// TIA Portal V16 export
// export: Created 2022-08-03T14:37:58.543671Z, ExportSetting WithDefaults, DisplayName Totally Integrated Automation Portal, DisplayVersion V16, DisplayName TIA Portal Version Control Interface, DisplayVersion V16, DisplayName TIA Portal Openness, DisplayVersion V16, DisplayName SINAMICS Startdrive Advanced, DisplayVersion V16, DisplayName SINAMICS Startdrive G130, G150, S120, S150, SINAMICS MV, S210, DisplayVersion V16, DisplayName SINAMICS Startdrive G110M, G120, G120C, G120D, G120P, DisplayVersion V16, DisplayName STEP 7 Professional, DisplayVersion V16, DisplayName STEP 7 Safety, DisplayVersion V16, DisplayName WinCC Professional, DisplayVersion V16
ORGANIZATION_BLOCK "Electrical_interlock"   // OB1, LAD, ProgramCycle
TITLE = "Main Program Sweep (Cycle)"
{ S7_Optimized_Access := 'TRUE' }
VERSION : 0.1
// stored: AutoNumber true, IsIECCheckEnabled false, SetENOAutomatically false
   VAR_INPUT
      Initial_Call : Bool;   // Initial call of this OB
      Remanence : Bool;   // =True, if remanent data are available
   END_VAR
BEGIN

REGION Network 1
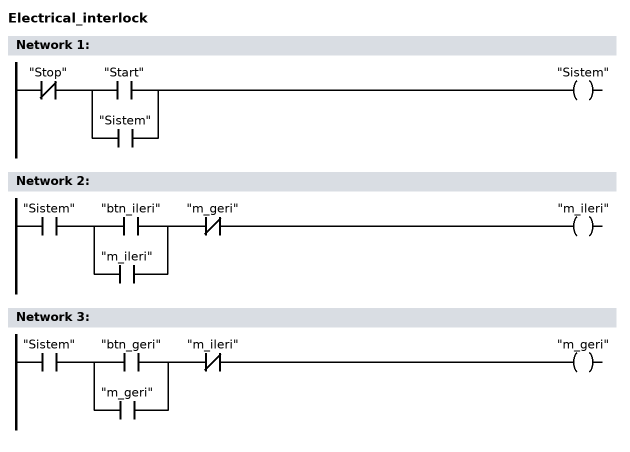
   RUNG wire#powerrail
      I_Contact( "Stop" )
      wire#w1
      Contact( "Start" )
      wire#w2
      Coil( "Sistem" )
   END_RUNG
   RUNG wire#w1
      Contact( "Sistem" )
   END_RUNG wire#w2
   // the same network as SCL:
   "Sistem" := NOT "Stop" AND ("Start" OR "Sistem");
END_REGION

REGION Network 2
   RUNG wire#powerrail
      Contact( "Sistem" )
      wire#w1
      Contact( "btn_ileri" )
      wire#w2
      I_Contact( "m_geri" )
      Coil( "m_ileri" )
   END_RUNG
   RUNG wire#w1
      Contact( "m_ileri" )
   END_RUNG wire#w2
   // the same network as SCL:
   "m_ileri" := "Sistem" AND ("btn_ileri" OR "m_ileri") AND NOT "m_geri";
END_REGION

REGION Network 3
   RUNG wire#powerrail
      Contact( "Sistem" )
      wire#w1
      Contact( "btn_geri" )
      wire#w2
      I_Contact( "m_ileri" )
      Coil( "m_geri" )
   END_RUNG
   RUNG wire#w1
      Contact( "m_geri" )
   END_RUNG wire#w2
   // the same network as SCL:
   "m_geri" := "Sistem" AND ("btn_geri" OR "m_geri") AND NOT "m_ileri";
END_REGION
END_ORGANIZATION_BLOCK
